{attribute 'pack_mode' := '2'}
TYPE ST_CAM_STATE :
STRUCT
  nNumPointsRead          : UDINT;

END_STRUCT
END_TYPE

(* stored: Version 1.1.0.1, ProductVersion 3.1.4024.12
   DUT ST_CAM_STATE: Id {429d5f47-2b73-0837-3eef-3bb02acbf2ef} *)
